// TIA Portal V20 export
DATA_BLOCK "DB_Xml"   // DB7
{ S7_Optimized_Access := 'TRUE' }
   VAR
      Speed : Real := 2.5;
      Mode : Int;
   END_VAR
BEGIN
END_DATA_BLOCK
